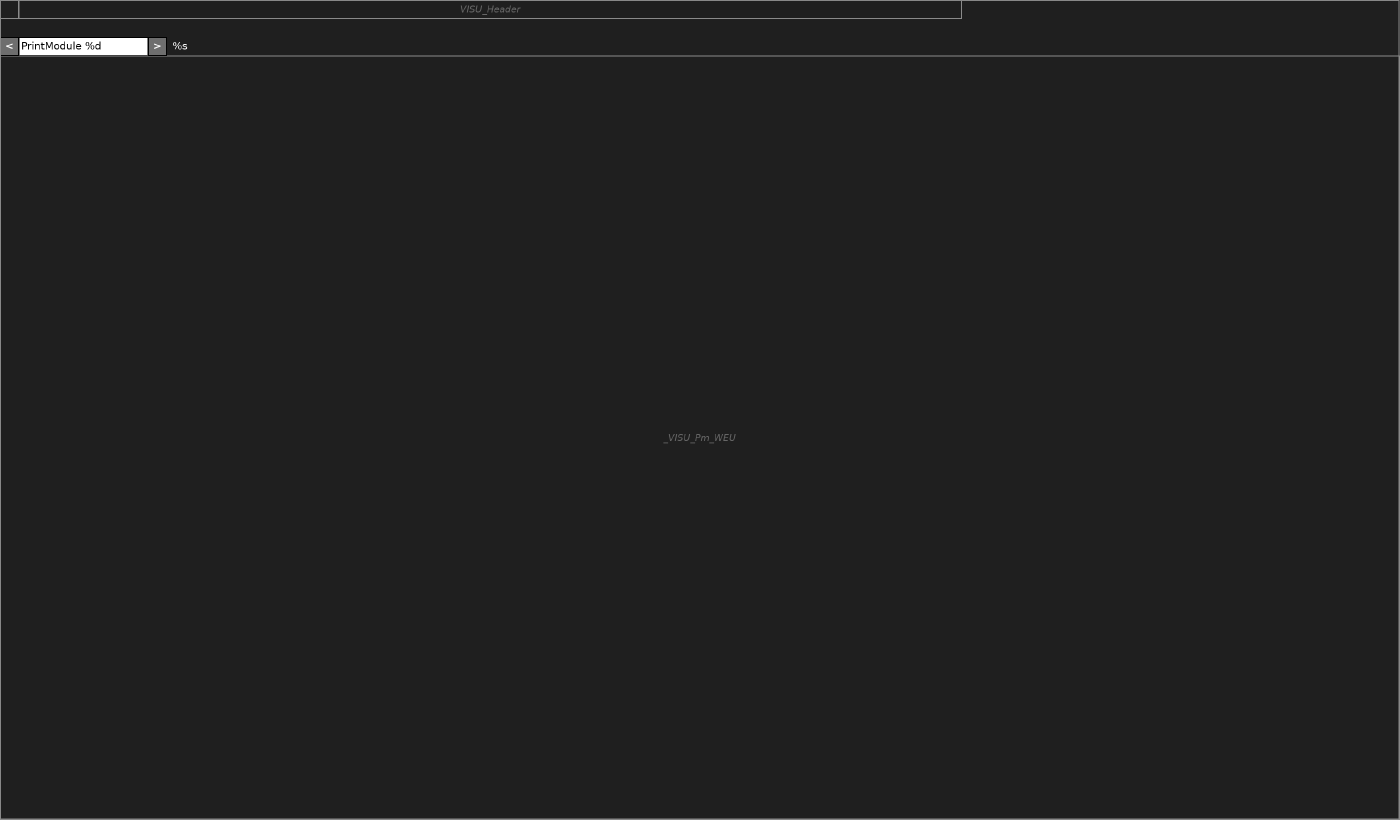
VISUALIZATION VISU_PrintModule_Detail  // 1514x887
    Rectangle (20,40 140x20), "PrintModule %d", text variable: PRG_PRINT.fbModuleMaster.nViewPmSel
    Frame (0,60 1514x827)
        shows _VISU_Pm_WEU(mInst := PRG_PRINT.fbPrintModule[PRG_PRINT.fbModuleMaster.nViewPmSel])
    Frame (20,0 1020x20)
        shows VISU_Header()
    Frame (0,0 20x20)
        shows VISU_ButtonBack()
    RoundedRectangle (160,40 20x20), ">"
        OnMouseClick: execute { PRG_PRINT.fbModuleMaster.nViewPmSel := PRG_PRINT.fbModuleMaster.nViewPmSel + 1; }
    RoundedRectangle (0,40 20x20), "<"
        OnMouseClick: execute { PRG_PRINT.fbModuleMaster.nViewPmSel := PRG_PRINT.fbModuleMaster.nViewPmSel - 1; }
    Rectangle (180,40 300x20), "%s", text variable: PRG_PRINT.fbModuleMaster._sModules[PRG_PRINT.fbModuleMaster.nViewPmSel]^._instanceName
END_VISUALIZATION

(* stored: Version 1.1.0.1, ProductVersion 3.1.4024.11
   Visu VISU_PrintModule_Detail: Id {cefb1ae0-691a-4fb5-812f-b682a2a54c9e} *)
